# EPICS autosave request: es-vortex/auto_settings.req
file "dxpSystem_settings.req",          P=$(P)
file "dxpSaturn_settings.req",          P=$(P)
file "dxpHighLevel_settings.req",       P=$(P), R=dxp1:
file "mca_settings.req",                P=$(P), M=mca1
